FUNCTION_BLOCK ABSTRACT Xts IMPLEMENTS ICyclic, I_Initialise
VAR
	MyName : STRING;
	_MyXts : INT;
	_XtsEnabled : BOOL;
	XtsIoEnvVar : XTSIOEnvVarWrapper;
	mcCollisionGroup : CollisionGroup;
	XtsHardware : XTSHardware := (MyXtsIoEnvVarWrapper := XtsIoEnvVar);
	XtsHwState : XtsSystemInitialisation;
	EnableSequence : XtsEnableSequence(mcCollisionGroup);
	DisableSequence : XtsDisableSequence(mcCollisionGroup);
	State : UINT;	
	i : UINT;
	AtHome: BOOL;
	EnabledTrigger : R_TRIG;
	DisabledTrigger : R_TRIG;
END_VAR
VAR_IN_OUT
	_MoverArray : ARRAY[*] OF ITF_XtsMoverAxis;
END_VAR

{analysis -2}

METHOD PUBLIC ActivateTracksInMovers : BOOL
VAR
	ActivateTrackResult : BOOL;
END_VAR
FOR i := 1 TO TO_UINT(UPPER_BOUND(_MoverArray,1)) DO
	_MoverArray[i].ActivateTrack(newTrack := _MoverArray[i].MoversActiveTrack,
									Track := XtsHardware.GetTrackByOTCID(trackOTCID := _MoverArray[i].MoversActiveTrack));
END_FOR
ActivateTracksInMovers := true;
END_METHOD

METHOD PUBLIC Cycle : HRESULT
VAR
	EnableResult : HRESULT;
	DisableResult : HRESULT;
	GrpStopResult : HRESULT;
	CollisionResult : HRESULT;
END_VAR
EnableResult := EnableSequence.Cycle();
DisableResult := DisableSequence.Cycle();
CollisionResult := mcCollisionGroup.Cycle();
EnabledTrigger(CLK := EnableSequence.Done);
DisabledTrigger(CLK := DisableSequence.Done);
XtsHardware.Cycle();
IF EnabledTrigger.Q THEN
	_XtsEnabled := TRUE;
END_IF
IF DisabledTrigger.Q THEN
	_XtsEnabled := false;
END_IF
IF EnableResult = E_FAIL OR
	DisableResult = E_FAIL OR
	GrpStopResult = E_FAIL OR
	CollisionResult = E_FAIL THEN
	Cycle := E_FAIL;
END_IF
END_METHOD

METHOD DisableXTS : BOOL
VAR_INPUT
END_VAR
DisableXTS := DisableSequence.Disable();
END_METHOD

METHOD EnableXTS : BOOL
VAR_INPUT
END_VAR
EnableSequence.Enable();
END_METHOD

METHOD PUBLIC GetTMSMoverInterface : BOOL
VAR_INPUT
END_VAR
VAR
END_VAR
FOR i := 1 TO TO_UINT(UPPER_BOUND(_MoverArray,1)) DO
	_MoverArray[i].MoverXtsIoEnvInterface := XtsIoEnvVar.GetMoverInterface(i);
END_FOR
END_METHOD

METHOD GetTrackByOCTID : I_XtsTrack
VAR_INPUT
	TrackId : OTCID;
END_VAR
GetTrackByOCTID := XtsHardware.GetTrackByOTCID(trackOTCID := TrackId);
END_METHOD

METHOD Initialise : HRESULT
VAR_INPUT
END_VAR
CASE XtsHwState OF
	XtsSystemInitialisation.Init:
		IF XtsIoEnvVar.Initialise() THEN
			XtsHwState := XtsSystemInitialisation.PassGroupReference;
		END_IF
		
	XtsSystemInitialisation.PassGroupReference:
		mcCollisionGroup.CAGroupXtsIoEnvInterface := XtsIoEnvVar.GetCaGroupInterface(_MyXts);
		XtsHwState := XtsSystemInitialisation.InitialiseHardware;
	
	XtsSystemInitialisation.InitialiseHardware:
		IF XtsHardware.Initialise() = 2 THEN
			MyName := XtsHardware.MyName;
			XtsHwState := XtsSystemInitialisation.SetDetection;
		END_IF
	
	XtsSystemInitialisation.SetDetection:
		IF XtsHardware.SetTrackForDetection(1) THEN
			XtsHwState := XtsSystemInitialisation.Redetect;
		END_IF
		
	XtsSystemInitialisation.Redetect:
		IF XtsHardware.TriggerMoverDetection() THEN
			XtsHwState := XtsSystemInitialisation.MoversValid;
		END_IF
		
	XtsSystemInitialisation.MoversValid:
		IF XtsHardware.getAllMoversValid() THEN
			XtsHwState := XtsSystemInitialisation.AllMoversFound;
		END_IF
	
	XtsSystemInitialisation.AllMoversFound:
		IF XtsHardware.getMoversDetected() THEN
			XtsHwState := XtsSystemInitialisation.XTSMode;
		END_IF
		
	XtsSystemInitialisation.XTSMode:
		IF XtsHardware.IsInSim() THEN
			XtsHwState := XtsSystemInitialisation.MoverIdDetection;
		ELSE
			XtsHwState := XtsSystemInitialisation.CheckModuleVoltages;
		END_IF
		
	XtsSystemInitialisation.CheckModuleVoltages:
		IF XtsHardware.Is24VdcOK() = 2 AND XtsHardware.Is48VdcOK() = 2 THEN
			XtsHwState := XtsSystemInitialisation.MoverIdDetection;
		END_IF
	
	XtsSystemInitialisation.MoverIdDetection:
		IF XtsHardware.TriggerMoverID() THEN
			XtsHwState := XtsSystemInitialisation.HWReady;
			GetTMSMoverInterface();
		END_IF
	
	XtsSystemInitialisation.HWReady:
		Initialise := 2;	
END_CASE
END_METHOD

METHOD IsXtsIdle : BOOL
VAR_INPUT
END_VAR
IsXtsIdle := DisableSequence.Done;
END_METHOD

METHOD IsXtsReady : BOOL
VAR_INPUT
END_VAR
IsXtsReady := _XtsEnabled;
END_METHOD

METHOD PUBLIC Abstract MoverHomeSequence : BOOL
VAR_INPUT
END_VAR
END_METHOD

PROPERTY MyNumberOfParts : int
GET
MyNumberOfParts := XtsHardware.MyNumberParts;
END_GET
SET
XtsHardware.MyNumberParts := MyNumberOfParts;
END_SET
END_PROPERTY

PROPERTY MyNumberOfTracks : int
GET
MyNumberOfTracks := XtsHardware.MyNumberTracks;
END_GET
SET
XtsHardware.MyNumberTracks := MyNumberOfTracks;
END_SET
END_PROPERTY

PROPERTY MyXts : INT
GET
MyXts := XtsHardware.MyXts;
END_GET
SET
XtsHardware.MyXts := _MyXts := MyXts;
END_SET
END_PROPERTY

METHOD StopXts : BOOL
VAR_INPUT
END_VAR
mcCollisionGroup.GroupStop();
END_METHOD

END_FUNCTION_BLOCK

(* stored: Version 1.1.0.1
   POU Xts: Id {4538c683-94fc-49a1-b5ad-30ffec5e4eff}, SpecialFunc None
   Folder Operations: Id {0e8598c4-3d58-4c14-a12f-6fd3f3ea02bf}
   Folder Settings: Id {cec05bdb-9232-4b5d-b91e-848bd7bc55d9}
   Folder Status: Id {c34f5481-c408-4671-a299-9c4a6e31956c}
   Method ActivateTracksInMovers: Id {682f2d4e-bf73-44bf-93e3-716a6d45755c}
   Method Cycle: Id {da42838e-fb00-40a5-96f4-b787aa883566}
   Method DisableXTS: Id {e2a85e5a-c7bf-481d-be4f-81acebc29fb7}
   Method EnableXTS: Id {e800781e-1435-4747-9cb4-9b9fab34ca22}
   Method GetTMSMoverInterface: Id {0e64eced-3444-47ea-9660-c818e7a9dea9}
   Method GetTrackByOCTID: Id {1d75e1be-3c32-4213-9fda-cb384fa7a069}
   Method Initialise: Id {3c52ae7d-89c5-4979-a1bd-5023a279947c}
   Method IsXtsIdle: Id {98f4e7e8-94b6-4461-9a7b-2bd1c0aafde4}
   Method IsXtsReady: Id {73e2c3f0-1b32-45c2-a8cc-fbf01ac18258}
   Method MoverHomeSequence: Id {5c2deb91-ebd0-4a93-99ec-6a6bbbd5e076}
   Property MyNumberOfParts: Id {33632734-2180-4c77-982d-f6997ead5bb5}
   Get Get: Id {ec285ff9-810a-46b0-8941-68dcdc1ab79d}
   Set Set: Id {4cb5fde4-6845-43ef-b95e-df4929829b0c}
   Property MyNumberOfTracks: Id {6b69c4c6-afe3-46d9-bc08-86224f82f24a}
   Get Get: Id {cab0d03f-ccb1-4d2e-adb6-3d697ceee44c}
   Set Set: Id {b24fc04c-e333-4935-bdff-3eff5a7d9932}
   Property MyXts: Id {b982f888-fcea-49f3-8b85-76339b257fce}
   Get Get: Id {7260ae55-6d72-4286-9779-c205f4bf658b}
   Set Set: Id {f9bbe24a-eac8-4b47-a949-a650212b0818}
   Method StopXts: Id {4b648283-f5f4-4d47-a58f-be53e519365d} *)
